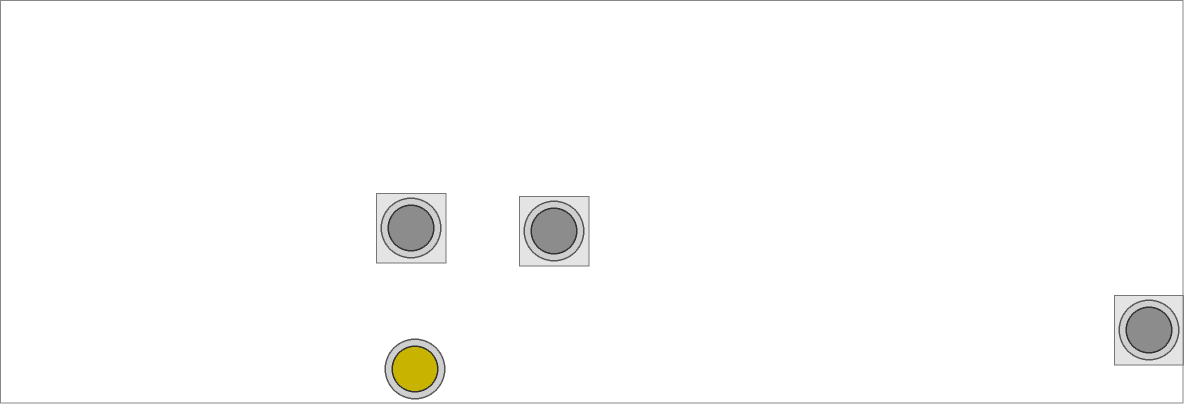
VISUALIZATION Visualization  // 1184x404
    Lamp1 (380,334 70x70), variable: GVL.LED_BestellingGeplaatst, style: Lamp-Lamp1-Yellow
    PushSwitch (519,196 70x70), variable: GVL.BT_Deurbel, behaviour: TAP, style: Switch-PushSwitch-Gray
    PushSwitch (1114,295 70x70), variable: GVL.Reset, behaviour: TAP, style: Switch-PushSwitch-Gray
    PushSwitch (376,193 70x70), variable: GVL.BT_BestellingPlaatsen, behaviour: TAP, style: Switch-PushSwitch-Gray
END_VISUALIZATION

(* stored: Version 1.1.0.1, ProductVersion 3.1.4024.13
   Visu Visualization: Id {d9f129e3-21d9-476c-99fc-234acaa998e8} *)
